PROGRAM p_XLegacyPLCModbus
VAR
	fbHXX_PLCInputCoilsRx	:	FB_MBReadCoils;
	fbXCS_PLCInputCoilsRx	:	FB_MBReadCoils;
	
	i_xHXX_PLC_CnBits	:	ARRAY [0..20] OF BYTE;
	i_xXCS_PLC_CnBits	:	ARRAY [0..20] OF BYTE;
	
	ftResetHXX	: F_TRIG; 
	ftResetXCS	: F_TRIG; 
	tonRetryHXX	: TON;
	tonRetryXCS : TON;
END_VAR


(* Modbus Info for Koyo
Modbus Addresses for
Koyo DL05/06/240/250/260/430/440/450 PLCs
PLC Memory Type		| Modbus start address Decimal (octal) | Function codes
Inputs (X)			  2048 (04000)							2
Special Relays (SP)	  3072 (06000)							2
Outputs (Y)			  2048 (04000)							1, 5, 15
Control Relays (C)	  3072 (06000)							1, 5, 15
Timer Contacts (T)	  6144 (014000)							1, 5, 15
Counter Contacts (CT) 6400 (014400)							1, 5, 15
Stage Status Bits (S) 6144 (012000)							1, 5, 15
*)

(* HXX code *)

// Retry after some time
tonRetryHXX.IN := NOT fbHXX_PLCInputCoilsRx.bBusy;
tonRetryHXX.PT := T#10S;
tonRetryHXX();

ftResetHXX(CLK:=fbHXX_PLCInputCoilsRx.bBusy);
ftResetHXX();

fbHXX_PLCInputCoilsRx.bExecute := ftResetHXX.Q OR tonRetryHXX.Q;

fbHXX_PLCInputCoilsRx(sIPAddr:='172.21.36.66', nTCPPort:=502, nQuantity:=32, nMBAddr:=8#6000, cbLength:=SIZEOF(i_xHXX_PLC_CnBits),  pDestAddr:=ADR(i_xHXX_PLC_CnBits), tTimeout:=T#10S);

IF fbHXX_PLCInputCoilsRx.bError THEN
	//run some error code for modbus
	//if there's a modbus error, set all incoming bits to zero, set 
	// HXX PLC Relay coil C[10] is used for MXT:GCC:06.VacOK
	i_xHXX_PLC_CnBits[0].0 := 0;
	i_xHXX_PLC_CnBits[0].1 := 0;
	i_xHXX_PLC_CnBits[0].2 := 0;
	i_xHXX_PLC_CnBits[0].3 := 0;
	i_xHXX_PLC_CnBits[0].4 := 0;
	i_xHXX_PLC_CnBits[1].0 := 0;
	i_xHXX_PLC_CnBits[1].1 := 0;
	i_xHXX_PLC_CnBits[1].2 := 0;
	
	
	
ELSIF ftResetHXX.Q AND fbHXX_PLCInputCoilsRx.cbRead > 0 THEN
	fbHXX_PLCInputCoilsRx.bExecute := FALSE;
	
	//i_xUSVacOK := i_xHXX_PLC_CnBits[1].0;
	
ELSIF fbHXX_PLCInputCoilsRx.cbRead = 0 THEN
			//more error code cause we didn't manage to read anything
			//i_xUSVacOK := FALSE;
			g_xNoHXXPLCResponse:= TRUE;
			
END_IF
 
(* XCS code *)
tonRetryXCS.IN := NOT fbXCS_PLCInputCoilsRx.bBusy;
tonRetryXCS.PT := T#10S;
tonRetryXCS();

ftResetXCS(CLK:=fbXCS_PLCInputCoilsRx.bBusy);
ftResetXCS();

fbXCS_PLCInputCoilsRx.bExecute := ftResetXCS.Q OR tonRetryXCS.Q;

fbXCS_PLCInputCoilsRx(sIPAddr:='172.21.43.73', nTCPPort:=502, nQuantity:=32, nMBAddr:=8#6000, cbLength:=SIZEOF(i_xXCS_PLC_CnBits),  pDestAddr:=ADR(i_xXCS_PLC_CnBits), tTimeout:=T#10S);

IF fbXCS_PLCInputCoilsRx.bError THEN
	//run some error code for modbus
	//if there's a modbus error, set all incoming bits to zero
	// XCS PLC Relay coil?
	i_xXCS_PLC_CnBits[0].0 := 0;
	i_xXCS_PLC_CnBits[0].1 := 0;
	i_xXCS_PLC_CnBits[0].2 := 0;
	i_xXCS_PLC_CnBits[0].3 := 0;
	i_xXCS_PLC_CnBits[0].4 := 0;
	i_xXCS_PLC_CnBits[1].0 := 0;
	i_xXCS_PLC_CnBits[1].1 := 0;
	i_xXCS_PLC_CnBits[1].2 := 0;
	
	
	
ELSIF ftResetXCS.Q AND fbXCS_PLCInputCoilsRx.cbRead > 0 THEN
	fbXCS_PLCInputCoilsRx.bExecute := FALSE;
	//q_xDSVacOK := i_xXCS_PLC_CnBits[1].0;
	
ELSIF fbXCS_PLCInputCoilsRx.cbRead = 0 THEN
			//more error code cause we didn't manage to read anything
			g_xDSVacOK := FALSE;
			g_xNoXCSPLCResponse:= TRUE;
			
END_IF


(* // Retry after some time
	tonRetry.IN := NOT fbSXRPLCInputCoilsRx.bBusy;
	tonRetry.PT := T#10S;
	tonRetry();
	
	ftResetHXX.CLK:=fbSXRPLCInputCoilsRx.bBusy;
	ftResetHXX();
	
	fbSXRPLCInputCoilsRx.bExecute := ftResetHXX.Q OR tonRetry.Q;
	
	IF fbSXRPLCInputCoilsRx.bError THEN
		//run some error code for modbus
		//if there's a modbus error, set all incoming bits to zero
		g_xUpstreamVacOK := FALSE;
		g_xNoPLCResponse:= FALSE;
	ELSIF ftResetHXX.Q THEN
		IF fbSXRPLCInputCoilsRx.cbRead > 0 THEN
			g_xUpstreamVacOK := i_xSXRPLC_CnBits[1].0;
			g_xNoPLCResponse:= FALSE;
			
		ELSIF fbSXRPLCInputCoilsRx.cbRead = 0 THEN
			//more error code cause we didn't manage to read anything
			g_xUpstreamVacOK := FALSE;
			g_xNoPLCResponse:= TRUE;
		END_IF
	ELSE
		;
	END_IF
	
	fbSXRPLCInputCoilsRx(sIPAddr:='172.21.39.48', nTCPPort:=502, 
						nQuantity:=10, nMBAddr:=8#6000, cbLength:=SIZEOF(i_xSXRPLC_CnBits), pDestAddr:=ADR(i_xSXRPLC_CnBits), 
						tTimeout:=T#10S);
						
	//reset lamp values
	i_xLAMPPLC_InputCoils := 0; *)

END_PROGRAM

(* stored: Version 1.1.0.1, ProductVersion 3.1.4020.12
   POU p_XLegacyPLCModbus: Id {a477c376-dd06-40c3-b569-438369655d9b}, SpecialFunc None *)
